TYPE (* IEC61131-3, Table 14#5 *)
  (* Standard: 1131-3 *)
  (* Version 0.0, 10/1/2026, Schneider Electric, Template *)
  PACKAGE Main;
  {SET_ATTRIBUTE(nxtDataType, CFRnm49gOBxVMwHd2RMQBFf+UJjqvPlP5l9jCDo0iCxmhRDl9zNqgQ==)}
  dtRange : INT(0..100);
END_TYPE
